KUKA KRL program: tip_change.src, tip_change.dat

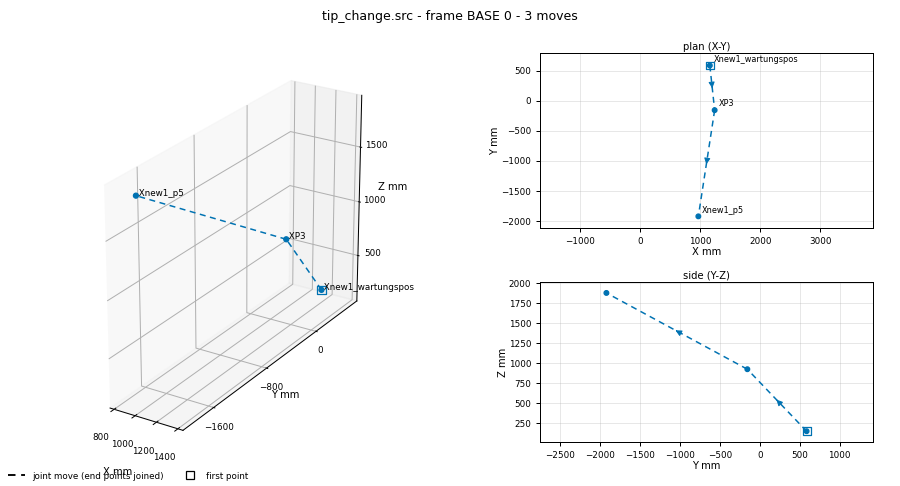
[picture p0: tool path of tip_change.src in frame BASE 0, 3 of 7 moves have a stored position in this frame; points joined in program order, loops and branches not executed]
--- tip_change.src ---
&ACCESS RVO1
&REL 51
&PARAM DISKPATH = KRC:\R1\Program\Outros
DEF TIP_CHANGE ( )
;FOLD INI;%{PE}
  ;FOLD BASISTECH INI
    GLOBAL INTERRUPT DECL 3 WHEN $STOPMESS==TRUE DO IR_STOPM ( )
    INTERRUPT ON 3
    BAS (#INITMOV,0 )
  ;ENDFOLD (BASISTECH INI)
;FOLD SPOTTECH INI
USERSPOT(#INIT)
;ENDFOLD (SPOTTECH INI)
;FOLD GRIPPERTECH INI
USER_GRP(0,DUMMY,DUMMY,GDEFAULT)
;ENDFOLD (GRIPPERTECH INI)
  ;FOLD USER INI
    ;Make your modifications here

  ;ENDFOLD (USER INI)
;ENDFOLD (INI)

; Caracterização dos meios de produção:
; Versão Atual:
; 04/05/2013 12:00 Name: P13.090-R6 CHANGES: Troca de capa

;FOLD PTP HOME Vel=100 % DEFAULT;%{PE}%R 8.2.24,%MKUKATPBASIS,%CMOVE,%VPTP,%P 1:PTP, 2:HOME, 3:, 5:100, 7:DEFAULT
$BWDSTART=FALSE
PDAT_ACT=PDEFAULT
FDAT_ACT=FHOME
BAS(#PTP_PARAMS,100)
$H_POS=XHOME
PTP XHOME
;ENDFOLD

CHK_W1_Wechs_OK ( )          ; CHECK C1 OK

;FOLD OUT 3218 'SPECIAL-POSITION REACHED' State=FALSE ;%{PE}%R 8.2.24,%MKUKATPBASIS,%COUT,%VOUTX,%P 2:3218, 3:SPECIAL-POSITION REACHED, 5:FALSE, 6:
$OUT[3218]=FALSE
;ENDFOLD
;FOLD WAIT FOR ( IN 3218 'REQUEST SPECIAL-POSITION' );%{PE}%R 8.2.24,%MKUKATPBASIS,%CEXT_WAIT_FOR,%VEXT_WAIT_FOR,%P 2:, 4:, 5:$IN, 6:3218, 7:REQUEST SPECIAL-POSITION, 9:
WAIT FOR  ( $IN[3218] )
;ENDFOLD

;FOLD PTP P1 Vel=100 % PDAT1 Tool[1]:Gun C1 Base[1]:Actros;%{PE}%R 8.2.24,%MKUKATPBASIS,%CMOVE,%VPTP,%P 1:PTP, 2:P1, 3:, 5:100, 7:PDAT1
$BWDSTART=FALSE
PDAT_ACT=PPDAT1
FDAT_ACT=FP1
BAS(#PTP_PARAMS,100)
PTP XP1
;ENDFOLD
;FOLD PTP P2 CONT Vel=100 % PDAT2 Tool[1]:Gun C1 Base[1]:Actros;%{PE}%R 8.2.24,%MKUKATPBASIS,%CMOVE,%VPTP,%P 1:PTP, 2:P2, 3:C_PTP, 5:100, 7:PDAT2
$BWDSTART=FALSE
PDAT_ACT=PPDAT2
FDAT_ACT=FP2
BAS(#PTP_PARAMS,100)
PTP XP2 C_PTP
;ENDFOLD

;FOLD PTP new1_wartungspos  Vel=100 % P_OLP3 Tool[1]:Gun C1 Base[0];%{PE}%R8.3,%MKUKATPBASIS,%CMOVE,%VPTP,%P 1:PTP, 2:new1_wartungspos, 3:, 5:100, 7:P_OLP3
$BWDSTART = FALSE
PDAT_ACT= PP_OLP3
FDAT_ACT= Fnew1_wartungspos
BAS(#PTP_PARAMS,100)
PTP Xnew1_wartungspos
;ENDFOLD

;FOLD OUT 3218 'SPECIAL-POSITION REACHED' State=TRUE ;%{PE}%R 8.2.24,%MKUKATPBASIS,%COUT,%VOUTX,%P 2:3218, 3:SPECIAL-POSITION REACHED, 5:TRUE, 6:
$OUT[3218]=TRUE
;ENDFOLD
Halt
;FOLD WAIT FOR ( NOT IN 3218 'REQUEST SPECIAL-POSITION' );%{PE}%R 8.2.24,%MKUKATPBASIS,%CEXT_WAIT_FOR,%VEXT_WAIT_FOR,%P 2:, 4:NOT, 5:$IN, 6:3218, 7:REQUEST SPECIAL-POSITION, 9:
WAIT FOR  (  NOT $IN[3218] )
;ENDFOLD

;FOLD PTP P3 CONT Vel=100 % PDAT3 Tool[1]:Gun C1 Base[0];%{PE}%R 8.2.24,%MKUKATPBASIS,%CMOVE,%VPTP,%P 1:PTP, 2:P3, 3:C_PTP, 5:100, 7:PDAT3
$BWDSTART=FALSE
PDAT_ACT=PPDAT3
FDAT_ACT=FP3
BAS(#PTP_PARAMS,100)
PTP XP3 C_PTP
;ENDFOLD

;FOLD ; Teste de solda;%{PE}%R 8.2.24,%MKUKATPBASIS,%CCOMMENT,%VNORMAL,%P 2:Teste  de  solda
;ENDFOLD
;FOLD PTP new1_p5 P_OLP5 SPOT Gun=1 RETR OPN S_OLP1;%{PE}%R8.3,%MKUKATPSPOT,%CSPOT,%VPTP,%P 1:PTP, 2:new1_p5, 3:, 5:100, 7:P_OLP5, 10:1, 12:0, 14:#OPN, 16:1, 18:0, 20:0.0, 22: 0.0, 24: 1, 25:S_OLP1
PDAT_ACT= PP_OLP5
BAS(#PTP_DAT)
FDAT_ACT= Fnew1_p5
BAS(#FRAMES)
BAS(#VEL_PTP,100)
S_ACT.GUN=1
S_ACT.PAIR=SDEFAULT.PAIR
S_ACT.RETR=#OPN
S_ACT.CLO_TM=SS_OLP1.CLO_TM
S_ACT.PGNO1=SDEFAULT.PGNO1
S_ACT.PGNO2=SDEFAULT.PGNO2
S_ACT.PRESS1=SDEFAULT.PRESS1
S_ACT.PRESS2=SDEFAULT.PRESS2
S_READY=FALSE
USERSPOT(#ADVSPOT,S_ACT)
TRIGGER WHEN DISTANCE=1 DELAY=SS_OLP1.CLO_TM DO USERSPOT(#PRESPOT,S_ACT) PRIO=-1
TRIGGER WHEN DISTANCE=1 DELAY=0.0 DO USERSPOT(#SPOT,S_ACT) PRIO=-1
PTP Xnew1_p5
WAIT FOR S_READY
;ENDFOLD

;FOLD PTP HOME  Vel= 100 % DEFAULT;%{PE}%V3.2.0,%MKUKATPBASIS,%CMOVE,%VPTP,%P 1:PTP, 2:HOME, 3:, 5:100, 7:DEFAULT
$BWDSTART = FALSE
$H_POS=XHOME
PDAT_ACT=PDEFAULT
BAS (#PTP_DAT )
FDAT_ACT=FHOME
BAS (#FRAMES )
BAS (#VEL_PTP,100 )
PTP  XHOME
;ENDFOLD

;FOLD OUT 3218 'SPECIAL-POSITION REACHED' State=FALSE ;%{PE}%R 8.2.24,%MKUKATPBASIS,%COUT,%VOUTX,%P 2:3218, 3:SPECIAL-POSITION REACHED, 5:FALSE, 6:
$OUT[3218]=FALSE
;ENDFOLD
END

--- tip_change.dat ---
&ACCESS RVO1
&REL 51
&PARAM DISKPATH = KRC:\R1\Program\Outros
DEFDAT  tip_change
;FOLD EXTERNAL DECLARATIONS;%{PE}%MKUKATPBASIS,%CEXT,%VCOMMON,%P
;FOLD BASISTECH EXT;%{PE}%MKUKATPBASIS,%CEXT,%VEXT,%P
EXT  BAS (BAS_COMMAND  :IN,REAL  :IN )
DECL INT SUCCESS
;ENDFOLD (BASISTECH EXT)
;FOLD USER EXT;%{E}%MKUKATPUSER,%CEXT,%VEXT,%P
;Make your modifications here
;ENDFOLD (USER EXT)
;ENDFOLD (EXTERNAL DECLARATIONS)

;# ============ START PATH : tip_change =============
DECL FDAT Fnew1_p1={TOOL_NO 1,BASE_NO 0,IPO_FRAME #BASE,POINT2[] " "}
DECL PDAT PP_OLP1={VEL 100.0,ACC 100.0,APO_DIST 0.0}
DECL E6POS Xnew1_p1={X 2142.34204,Y 198.145996,Z 1881.30103,A 81.8957977,B 27.4578991,C -73.5851974,S 2,T 11}
DECL FDAT Fnew1_p7={TOOL_NO 1,BASE_NO 0,IPO_FRAME #BASE,POINT2[] " "}
DECL PDAT PP_OLP2={VEL 100.0,ACC 100.0,APO_DIST 0.0}
DECL E6POS Xnew1_p7={X 1156.27295,Y 423.039001,Z 383.427002,A 111.655296,B 2.09109998,C -2.08349991,S 2,T 10}
DECL FDAT Fnew1_wartungspos={TOOL_NO 1,BASE_NO 0,IPO_FRAME #BASE,POINT2[] " "}
DECL PDAT PP_OLP3={VEL 100.0,ACC 100.0,APO_DIST 0.0}
DECL E6POS Xnew1_wartungspos={X 1159.177,Y 587.393372,Z 148.890701,A 135.0495,B 2.68832493,C -0.445830196,S 18,T 11,E1 0.0,E2 0.0,E3 0.0,E4 0.0,E5 0.0,E6 0.0}
DECL FDAT Fnew1_p8={TOOL_NO 1,BASE_NO 0,IPO_FRAME #BASE,POINT2[] " "}
DECL PDAT PP_OLP4={VEL 100.0,ACC 100.0,APO_DIST 0.0}
DECL E6POS Xnew1_p8={X 1156.27295,Y 423.036987,Z 383.427002,A 111.655296,B 2.09109998,C -2.08340001,S 2,T 10}
DECL FDAT Fnew1_p5={TOOL_NO 1,BASE_NO 0,IPO_FRAME #BASE,POINT2[] " "}
DECL PDAT PP_OLP5={VEL 100.0,ACC 100.0,APO_DIST 0.0}
DECL SPOT_TYPE SS_OLP1={GUN 1,PAIR #FIRST,RETR #OPN,CLO_TM 1,PGNO1 1,PRESS1 0.0,PGNO2 0,PRESS2 0.0}
DECL E6POS Xnew1_p5={X 968.349426,Y -1921.25696,Z 1881.28699,A 13.3607302,B 27.4578209,C -73.5848236,S 18,T 10,E1 0.0,E2 0.0,E3 0.0,E4 0.0,E5 0.0,E6 0.0}
DECL FDAT Fnew1_p2={TOOL_NO 1,BASE_NO 0,IPO_FRAME #BASE,POINT2[] " "}
DECL PDAT PP_OLP6={VEL 100.0,ACC 100.0,APO_DIST 0.0}
DECL E6POS Xnew1_p2={X 2142.34204,Y 198.145996,Z 1881.30103,A 81.8957977,B 27.4578991,C -73.5851974,S 2,T 11}
DECL BASIS_SUGG_T LAST_BASIS={POINT1[] "P3                      ",POINT2[] "P3                      ",CP_PARAMS[] "CPDAT0                  ",PTP_PARAMS[] "PDAT3                   ",CONT[] "C_PTP                   ",CP_VEL[] "2.0                     ",PTP_VEL[] "100                     ",SYNC_PARAMS[] "SYNCDAT                 ",SPL_NAME[] "S0                      "}
DECL SPOT_SUGG_T LAST_SPOT={GUN[] " 1                      ",RETR_CMD[] "#OPN                    ",CHOISE[] "#FIRST                  ",CLO_TM[] "0                       ",PGNO1[] " 1                      ",PRESS1[] "0                       ",PGNO2[] " 1                      ",PRESS2[] "0                       ",SPOT_PARAMS[] "NORMAL                  "}
DECL E6POS XP1={X -2522.53711,Y 3934.45288,Z 1509.21802,A -166.4841,B 27.3574104,C -73.51474,S 18,T 10,E1 0.0,E2 0.0,E3 0.0,E4 0.0,E5 0.0,E6 0.0}
DECL FDAT FP1={TOOL_NO 1,BASE_NO 1,IPO_FRAME #BASE,POINT2[] " ",TQ_STATE FALSE}
DECL PDAT PPDAT1={VEL 100.0,ACC 100.0,APO_DIST 100.0,GEAR_JERK 50.0}
DECL E6POS XP2={X -2791.20801,Y 2166.323,Z 556.41803,A -83.9606781,B 13.1501703,C -3.9056499,S 18,T 10,E1 0.0,E2 0.0,E3 0.0,E4 0.0,E5 0.0,E6 0.0}
DECL FDAT FP2={TOOL_NO 1,BASE_NO 1,IPO_FRAME #BASE,POINT2[] " ",TQ_STATE FALSE}
DECL PDAT PPDAT2={VEL 100.0,ACC 100.0,APO_DIST 100.0,APO_MODE #CPTP,GEAR_JERK 50.0}
DECL E6POS XP3={X 1239.43005,Y -155.112595,Z 925.510925,A 95.9377213,B 13.2252102,C -3.81156802,S 18,T 10,E1 0.0,E2 0.0,E3 0.0,E4 0.0,E5 0.0,E6 0.0}
DECL FDAT FP3={TOOL_NO 1,BASE_NO 0,IPO_FRAME #BASE,POINT2[] " ",TQ_STATE FALSE}
DECL PDAT PPDAT3={VEL 100.0,ACC 100.0,APO_DIST 0.0,APO_MODE #CPTP,GEAR_JERK 50.0}
ENDDAT
